// TIA Portal V18 export
// export: Created 2025-12-01T12:38:06.9560666Z, ExportSetting None, DisplayName Totally Integrated Automation Portal, DisplayVersion V18 Update 5, DisplayName TIA Portal Openness, DisplayVersion V18 Update 5, DisplayName TIA Portal Teamcenter Gateway, DisplayVersion V18, DisplayName TIA Portal Version Control Interface, DisplayVersion V18, DisplayName STEP 7 Professional, DisplayVersion V18 Update 5, DisplayName STEP 7 Safety, DisplayVersion V18, DisplayName WinCC Professional, DisplayVersion V18 Update 5
DATA_BLOCK "PalletRelease"   // DB9001
{ S7_Optimized_Access := 'FALSE' }
// stored: AutoNumber false
   VAR
      Buffer : Struct
         AskPallet : Bool;
         UnloadFlag : Bool;
      END_STRUCT;
      LaserMarking : Struct
         AskPallet : Bool;
         UnloadFlag : Bool;
      END_STRUCT;
      Print : Struct
         AskPallet : Bool;
         UnloadFlag : Bool;
      END_STRUCT;
      Spare : Struct
         AskPallet : Bool;
         UnloadFlag : Bool;
      END_STRUCT;
      Spare2 : Struct
         AskPallet : Bool;
         UnloadFlag : Bool;
      END_STRUCT;
      "Time" : Array[0..1] of TOF_TIME;
      LaserMarkingBuffer : "LaserMarkingBuffer";
   END_VAR
BEGIN
END_DATA_BLOCK
